KUKA KRL program: chk_w4_grp2_opn.src

&ACCESS RVO2
&COMMENT Check GRP ACCELO Z2 OPEN
DEF chk_w4_grp2_opn( )

;//---- Start User-------
;Aguardando posicao de gripper fechado

$TIMER[10] = 0
$TIMER_STOP[10] = FALSE

WAIT FOR (NOT $IN[42] AND NOT $IN[44])
WAIT FOR ($IN[41] AND $IN[43])

$TIMER_STOP[10] = TRUE
$TIMER[10] = 0

;//---- End User-------
END
